TYPE CommonBlock_Struct :
UNION
		Value : INT;
		Bits : Bits_CommonBlock;
END_UNION
END_TYPE

(* stored: Version 1.1.0.1, ProductVersion 3.1.4022.18
   DUT CommonBlock_Struct: Id {b95a325b-578d-43af-9ee1-5c616130a699} *)
